FUNCTION_BLOCK _Template_Test EXTENDS TcUnit.FB_TestSuite
VAR
END_VAR

ExampleTest();

METHOD ExampleTest : BOOL
VAR
	expected : INT;
	actual : INT;
END_VAR
TcUnit.TEST('Example test');

expected := ;
actual := ;

AssertEquals(
	Expected := expected,
	Actual := actual,
	Message := 'What went wrong');

TEST_FINISHED();
END_METHOD

END_FUNCTION_BLOCK

(* stored: Version 1.1.0.1, ProductVersion 3.1.4024.12
   POU _Template_Test: Id {794ecc0f-2f93-47b7-aa99-433344a376da}, SpecialFunc None
   Method ExampleTest: Id {3dde4137-332e-41a2-9864-117beae40309} *)
